FUNCTION_BLOCK RingTokenSection (* Composite Function Block Type *)
  (* Standard: 61499-2 *)
  (* Version 0.2, 2003-12-05, JHC, Rockwell Automation, Renamed from NEWCOMPFB. *)
  (* Version 0.1, 2002-01-08, JHC, Rockwell Automation, Added DLY FB as example. *)
  (* Version 0.0, 2000-05-27, JHC, Rockwell Automation *)
  (* Compiler header: package fb.rt.cs725; *)
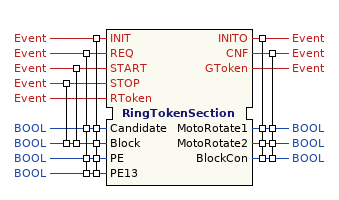
  EVENT_INPUT
    INIT WITH Candidate, Block, PE, PE13; (* Initialization Request *)
    REQ WITH Candidate, PE, PE13; (* Normal Execution Request *)
    START WITH Block;
    STOP WITH Block;
    RToken;
  END_EVENT
  EVENT_OUTPUT
    INITO WITH MotoRotate1, MotoRotate2, BlockCon; (* Initialization Confirm *)
    CNF WITH MotoRotate1, MotoRotate2, BlockCon; (* Execution Confirmation *)
    GToken;
  END_EVENT
  VAR_INPUT
    Candidate : BOOL;
    Block : BOOL;
    PE : BOOL;
    PE13 : BOOL;
  END_VAR
  VAR_OUTPUT
    MotoRotate1 : BOOL;
    MotoRotate2 : BOOL;
    BlockCon : BOOL;
  END_VAR
  FBS
    FC11 : ConveyorCTL(PE := 0, Block := 0, Candidate := 0);
    Conveyor4 : Conveyor_4;
  END_FBS
  EVENT_CONNECTIONS
    INIT TO FC11.INIT;
    REQ TO FC11.REQ;
    Conveyor4.INITO TO INITO;
    Conveyor4.CNF TO CNF;
    REQ TO Conveyor4.REQ;
    Conveyor4.STOP TO FC11.CAS_STOP;
    Conveyor4.START TO FC11.CAS_START;
    FC11.INITO TO Conveyor4.INIT;
    RToken TO Conveyor4.RToken;
    Conveyor4.GToken TO GToken;
  END_CONNECTIONS
  DATA_CONNECTIONS
    Block TO Conveyor4.Block;
    Candidate TO Conveyor4.Candidate;
    PE TO Conveyor4.PE;
    Conveyor4.BlockCon TO BlockCon;
    FC11.MotoRotate TO MotoRotate1;
    Conveyor4.MotoRotate TO MotoRotate2;
    PE13 TO Conveyor4.PE13;
  END_CONNECTIONS
END_FUNCTION_BLOCK
